FUNCTION F_StringCompNoCase : BOOL
VAR_INPUT
	s1		: STRING;
	s2		: STRING;
END_VAR
VAR
END_VAR


F_StringCompNoCase := ( F_ToUCase(s1) = F_ToUCase(s2) );

END_FUNCTION

(* stored: Version 1.1.0.1, ProductVersion 3.1.4024.5
   POU F_StringCompNoCase: Id {82af8c89-0c04-4ee4-b4d5-2be87f00b8e8}, SpecialFunc None *)
